// TwinCAT 3 PLC project PRG_B_HMIManager
// Title: B_HMIManager
// Company: RafałOS
// Author: Rafał Osajda
// ProjectVersion: 0.0.0.21
// ProgramVersion: 3.1.4024.0
// libraries:
//   B_Base, * (RafalOS)
//   B_Base_HMI_Connector, * (RafalOS)
//   B_HMIElements, * (RafalOS)
//   B_MachineControl, * (RafalOS)
//   B_MachineControl_HMI_Connector, * (RafalOS)
//   B_StatesAndModes, * (RafalOS)
//   Tc2_Standard, * (Beckhoff Automation GmbH)
//   Tc2_System, * (Beckhoff Automation GmbH)
//   Tc3_Module, * (Beckhoff Automation GmbH)
// project tree:
//   / PlcTask.TcTTO
//   POUs Compilation/ PRG_Compilation.TcPOU (not stored)
//   POUs/01_HMIManager/ FB_HMIManager.TcPOU, ITF_HMIManager.TcIO (not stored), ITF_HMIManagerConfigure.TcIO, ST_HMIManager.TcDUT
//   POUs/02_Configuration/ FB_HMIConfigure.TcPOU, ITF_HMIConfiguration.TcIO, ITF_HMIConfigure.TcIO (not stored)
// real-time tasks:
//   TASK PlcTask: cycle T#10ms, priority 20, ADS port 350

CONFIGURATION PRG_B_HMIManager
    RESOURCE PLC ON TwinCAT3
        TASK PlcTask(INTERVAL := T#10ms, PRIORITY := 20);
        PROGRAM PRG_Compilation WITH PlcTask : PRG_Compilation;
    END_RESOURCE
END_CONFIGURATION

// ---- POUs/01_HMIManager/ST_HMIManager.TcDUT
TYPE ST_HMIManager EXTENDS ST_BaseGroupElement_HMI_Link :
STRUCT
	stMainMenu			: ST_HMIEMenu_HMI_Link;
	stMachineControl	: ST_MCHMIMachineControl_HMI_Link;
	stRecipe			: ST_BaseRecipe_HMI;
END_STRUCT
END_TYPE

// ---- POUs/01_HMIManager/ITF_HMIManagerConfigure.TcIO
INTERFACE ITF_HMIManagerConfigure EXTENDS ITF_Base

(*			
	RafalOS
	Rafał Osajda		07.12.2025		TC 4024.66
	Dodawanie elementów do systemmu wyświetlania
*)
METHOD AddElementFromConfiguration
VAR_INPUT
	fbTopElementHMI		: ITF_BaseTopElement_HMI;
END_VAR
END_METHOD

(*			
	RafalOS
	Rafał Osajda		20.11.2025		TC 4024.66
	Dodawanie rozszerzonego wyświetlania danych inna prezenacja danych niż domyślna lista
*)
METHOD PUBLIC AddExtendedDisplayToPrepScrModuleFromConfiguration : BOOL
VAR_INPUT
	itfModule		: ITF_MCHMIPrepareDataForScreenExtension;
	itfExtension	: ITF_MCHMIDisplayExtension;
END_VAR
END_METHOD

(*			
	RafalOS
	Rafał Osajda		19.11.2025		TC 4024.66
	Dodanie połączenia do MachineControl  wywoływane z konfiguracji
*)
METHOD AddMachineControlConnectorFromConfiguration : BOOL
VAR_INPUT
	itfMachineControl	: ITF_MCHMIMachineControl_HMI;
END_VAR
END_METHOD

(*			
	RafalOS
	Rafał Osajda		14.11.2025		TC 4024.66
	Dodanie do systemu menu głównego 
*)
METHOD PUBLIC AddMainMenuFromConfiguration : BOOL
VAR_INPUT
	fbMenu			: ITF_HMIEMenu;
	fbMenu_HMI		: ITF_HMIEMenu_HMI;
END_VAR
END_METHOD

(*			
	RafalOS
	Rafał Osajda		19.11.2025		TC 4024.66
	Dodanie modułów do przygotowywania stron do wyświetlenia
*)
METHOD AddPrepareScreenModuleFromConfiguration : BOOL
VAR_INPUT
	itfModule	: ITF_MCHMIPrepareScreen_Init;
END_VAR
END_METHOD

(*			
	RafalOS
	Rafał Osajda		26.11.2025		TC 4024.66
	Podłaczenie modułu receptur
*)
METHOD PUBLIC AddRecipeModuleFromConfiguration : BOOL
VAR_INPUT
	fbRecipeModule		: ITF_BaseRecipe_HMI;
END_VAR
END_METHOD

METHOD PUBLIC GetNumberOfAddedButtons : INT
VAR_INPUT
END_VAR
END_METHOD

(*			
	RafalOS
	Rafał Osajda		18.11.2025		TC 4024.66
	Podłączenie głównej struktury danych dla domyślnych elementów 
*)
METHOD LinkHMIManagerDataFromConfiguration : BOOL
VAR_INPUT
	stData					: REFERENCE TO ST_HMIManager;
END_VAR
END_METHOD

METHOD PUBLIC LinkPrepareScreenToArrayFromConfiguration : BOOL
VAR_INPUT
	iScreen		: INT;
	iMode		: INT;
	itfModule	: ITF_MCHMIPrepareDataForScreen;
END_VAR
END_METHOD

(*			
	RafalOS
	Rafał Osajda		13.11.2025		TC 4024.66
	Podłączenie wsyzstkich zmiennych pochodzących od Programu safety 
*)
METHOD PUBLIC LinkSafetyToaddedElementsFromConfiguration : BOOL
VAR_INPUT
	flSS1				: ITF_BaseFlagGet;
	flSTO				: ITF_BaseFlagGet;
END_VAR
END_METHOD

(*			
	RafalOS
	Rafał Osajda		18.11.2025		TC 4024.66
	Ustawia przycisk na aktywny  - pierwsze okno w wyświetlaniu wizualizacji - wywoływane z konfiguracji
*)
METHOD SetButtonActiveFromConfiguration : BOOL
VAR_INPUT
	iNumber		: INT;	//numr przycisku
	bValue		: BOOL;
END_VAR
END_METHOD

(*			
	RafalOS
	Rafał Osajda		18.11.2025		TC 4024.66
	Ustawia przyciski na wlaczone lub wylaczone - możliwośc naciśnięcia
*)
METHOD SetButtonsEnabledFromConfiguration : BOOL
VAR_INPUT
	iNumber		: INT;	//numr przycisku
	bValue		: BOOL;
END_VAR
END_METHOD

(*			
	RafalOS
	Rafał Osajda		18.11.2025		TC 4024.66
	Ustawia przyciski na widoczne lub nie widoczne
*)
METHOD SetButtonsVisibleFromConfiguration : BOOL
VAR_INPUT
	iNumber		: INT;	//numr przycisku
	bValue		: BOOL;
END_VAR
END_METHOD

END_INTERFACE

// ---- POUs/02_Configuration/ITF_HMIConfiguration.TcIO
INTERFACE ITF_HMIConfiguration

(*			
	RafalOS
	Rafał Osajda		07.12.2025		TC 4024.66
	Dodawanie elementów do systemmu wyświetlania
*)
METHOD AddElement
VAR_INPUT
	itfHMIManager	: ITF_HMIManagerConfigure;
END_VAR
END_METHOD

(*			
	RafalOS
	Rafał Osajda		20.11.2025		TC 4024.66
	Dodawanie rozszerzonego wyświetlania danych inna prezenacja danych niż domyślna lista
*)
METHOD PUBLIC AddExtendedDisplayToPrepScrModule : BOOL
VAR_INPUT
	itfHMIManager	: ITF_HMIManagerConfigure;
END_VAR
END_METHOD

(*			
	RafalOS
	Rafał Osajda		19.11.2025		TC 4024.66
	Dodanie połączenia do MachineControl
*)
METHOD AddMachineControlConnector : BOOL
VAR_INPUT
	itfHMIManager	: ITF_HMIManagerConfigure;
END_VAR
END_METHOD

(*			
	RafalOS
	Rafał Osajda		14.11.2025		TC 4024.66
	Dodanie do systemu menu głównego 
*)
METHOD PUBLIC AddMainMenu : BOOL
VAR_INPUT
	itfHMIManager	: ITF_HMIManagerConfigure;
END_VAR
END_METHOD

(*			
	RafalOS
	Rafał Osajda		19.11.2025		TC 4024.66
	Dodanie modułów do przygotowywania stron do wyświetlenia
*)
METHOD AddPrepareScreenModule : BOOL
VAR_INPUT
	itfHMIManager	: ITF_HMIManagerConfigure;
END_VAR
END_METHOD

(*			
	RafalOS
	Rafał Osajda		26.11.2025		TC 4024.66
	Podłaczenie modułu receptur
*)
METHOD PUBLIC AddRecipeModule : BOOL
VAR_INPUT
	itfHMIManager	: ITF_HMIManagerConfigure;
END_VAR
END_METHOD

(*			
	RafalOS
	Rafał Osajda		18.11.2025		TC 4024.66
	Podłączenie głównej struktury danych dla domyślnych elementów 
*)
METHOD LinkHMIManagerData : BOOL
VAR_INPUT
	itfHMIManager	: ITF_HMIManagerConfigure;
END_VAR
END_METHOD

(*			
	RafalOS
	Rafał Osajda		16.12.2025		TC 4024.66
	Wywołanie linkowania zmiennych w topelemencie i jego dzieciach
*)
METHOD PUBLIC LinkMachineData : BOOL
VAR_INPUT
	itfHMIManager	: ITF_HMIManagerConfigure;
END_VAR
END_METHOD

(*			
	RafalOS
	Rafał Osajda		13.11.2025		TC 4024.66
	Podłączenie wsyzstkich zmiennych pochodzących od Programu safety 
*)
METHOD PUBLIC LinkSafetyToaddedElements : BOOL
VAR_INPUT
	itfHMIManager	: ITF_HMIManagerConfigure;
END_VAR
END_METHOD

(*			
	RafalOS
	Rafał Osajda		18.11.2025		TC 4024.66
	Ustawia przycisk na aktywny  - pierwsze okno w wyświetlaniu wizualizacji
*)
METHOD SetButtonActive : BOOL
VAR_INPUT
	itfHMIManager	: ITF_HMIManagerConfigure;
END_VAR
END_METHOD

(*			
	RafalOS
	Rafał Osajda		18.11.2025		TC 4024.66
	Ustawia przyciski na wlaczone lub wylaczone - możliwośc naciśnięcia
*)
METHOD SetButtonsEnabled : BOOL
VAR_INPUT
	itfHMIManager	: ITF_HMIManagerConfigure;
END_VAR
END_METHOD

(*			
	RafalOS
	Rafał Osajda		18.11.2025		TC 4024.66
	Ustawia przyciski na widoczne lub nie widoczne
*)
METHOD SetButtonsVisible : BOOL
VAR_INPUT
	itfHMIManager	: ITF_HMIManagerConfigure;
END_VAR
END_METHOD

END_INTERFACE

// ---- POUs/01_HMIManager/FB_HMIManager.TcPOU
FUNCTION_BLOCK FB_HMIManager EXTENDS FB_BaseGroupElement IMPLEMENTS ITF_HMIManager, ITF_HMIManagerConfigure
VAR
	(*	Inicjalizacja		*)
	bInitializeCycle			: BOOL;
	bInitDone					: BOOL;
	bIsValidData				: bool;
	(*	Konfiguracja		*)
	itfHMIConfigure				: ITF_HMIConfigure;		//moduł konfiguracji
	(*	Menu główne	*)
	itfMainMenu					: ITF_HMIEMenu;
	itfMainMenuHMI				: ITF_HMIEMenu_HMI;
	iNumberOfButtonMainMenu		: INT;
	iNumberOfActiveScreen		: INT;
	iNumberOfPreviewScreen		: INT;
	bChangePage					: BOOL;
//	(*	Obsługa zmiany strony	*)
//	arrChangePageSupport		: ARRAY [0..GVL_HMIEConstans.MAX_NUMBER_OF_BUTTON_IN_MENU] OF 
//									ARRAY [0..GVL_SaMConstans.NUMBER_OF_MODES] OF ITF_PrepareDataForScreen;
	(*	Dana wspólne dla całego systemu	*)
	refstManagerData			: REFERENCE TO ST_HMIManager;
	(*	Łącznik do MachineControl	*)
	itfMachineControl			: ITF_MCHMIMachineControl_HMI;
	(*	Lista dodanych elementów	*)
	stElement					: ST_ListOfElement_HMI;
END_VAR

IF (NOT THIS^.bInitializeCycle) THEN
	THIS^.bInitializeCycle		:= TRUE;
	THIS^.bInitDone				:= THIS^.InitializeCycle ();
ELSIF (THIS^.bInitDone) THEN
	THIS^.ExecuteCycle ();
END_IF

(*			
	RafalOS
	Rafał Osajda		07.12.2025		TC 4024.66
	Dodawanie elementów do systemmu wyświetlania
*)
METHOD AddElementFromConfiguration
VAR_INPUT
	fbTopElementHMI		: ITF_BaseTopElement_HMI;
END_VAR
fbTopElementHMI.JoinTheList (
	refstList		:= THIS^.stElement,
	iNumberOfParent := 0
);

fbTopElementHMI.LinkCommonData (stCommonData := THIS^.refstCommonData);
END_METHOD

(*			
	RafalOS
	Rafał Osajda		20.11.2025		TC 4024.66
	Dodawanie rozszerzonego wyświetlania danych inna prezenacja danych niż domyślna lista
*)
METHOD PUBLIC AddExtendedDisplayToPrepScrModuleFromConfiguration : BOOL
VAR_INPUT
	itfModule		: ITF_MCHMIPrepareDataForScreenExtension;
	itfExtension	: ITF_MCHMIDisplayExtension;
END_VAR
itfModule.LinkExtensionDisplay (fbExtendedDisplay := itfExtension);
END_METHOD

(*			
	RafalOS
	Rafał Osajda		19.11.2025		TC 4024.66
	Dodanie połączenia do MachineControl  wywoływane z konfiguracji
*)
METHOD AddMachineControlConnectorFromConfiguration : BOOL
VAR_INPUT
	itfMachineControl	: ITF_MCHMIMachineControl_HMI;
END_VAR
THIS^.itfMachineControl := itfMachineControl;

THIS^.itfMachineControl.LinkCommonData (stCommonData := THIS^.refstCommonData);
END_METHOD

(*			
	RafalOS
	Rafał Osajda		14.11.2025		TC 4024.66
	Dodanie do systemu menu głównego 
*)
METHOD PUBLIC AddMainMenuFromConfiguration : BOOL
VAR_INPUT
	fbMenu			: ITF_HMIEMenu;
	fbMenu_HMI		: ITF_HMIEMenu_HMI;
END_VAR
THIS^.SetText (eLocation := E_BaseLocation.pl, wsDescription := "Menu główne");
THIS^.SetText (eLocation := E_BaseLocation.en, wsDescription := "Main menu");
THIS^.SetText (eLocation := E_BaseLocation.de, wsDescription := "Hauptmenü");
fbMenu.SetName (stName := THIS^.GetTexts ());
THIS^.AddControlElement (itfControlElement := fbMenu);

THIS^.itfMainMenu := fbMenu;
THIS^.itfMainMenu.LinkCommonData (stCommonData := THIS^.refstCommonData);
//THIS^.itfMainMenu.LinkSS1 (fbSS1 := THIS^.itfSS1);
//THIS^.itfMainMenu.LinkSTO (fbSTO := THIS^.itfSTO);

THIS^.itfMainMenuHMI  := fbMenu_HMI;
THIS^.itfMainMenuHMI.LinkCommonData (stCommonData := THIS^.refstCommonData);
END_METHOD

(*			
	RafalOS
	Rafał Osajda		29.10.2025		TC 4024.66
	Dodawanie intefejsu konfiguracji
*)
METHOD PUBLIC AddModulConfigure : BOOL
VAR_INPUT
	fbHMIConfigure			: ITF_HMIConfigure;
END_VAR
THIS^.itfHMIConfigure		:= fbHMIConfigure;
END_METHOD

(*			
	RafalOS
	Rafał Osajda		19.11.2025		TC 4024.66
	Dodanie modułów do przygotowywania stron do wyświetlenia
*)
METHOD AddPrepareScreenModuleFromConfiguration : BOOL
VAR_INPUT
	itfModule	: ITF_MCHMIPrepareScreen_Init;
END_VAR
THIS^.itfMachineControl.AddPrepareScreenModuleFromManager (
	itfModule	:= itfModule
);
itfModule.LinkCommonData (stCommonData := THIS^.refstCommonData);
END_METHOD

(*			
	RafalOS
	Rafał Osajda		26.11.2025		TC 4024.66
	Podłaczenie modułu receptur
*)
METHOD PUBLIC AddRecipeModuleFromConfiguration : BOOL
VAR_INPUT
	fbRecipeModule		: ITF_BaseRecipe_HMI;
END_VAR
THIS^.itfMachineControl.AddRecipeModulFormManager (fbRecipeModul := fbRecipeModule);
END_METHOD

(*			
	RafalOS
	Rafał Osajda		10.11.2025		TC 4024.66
	Główna metoda sterujaca wyświetlaniem dsanych na HMI
*)
METHOD PUBLIC ExecuteCycle
	(* Testowanie MenuGlownego	*)
THIS^.itfMainMenu.Testing ();
	(*	Przepisanie Aktualnych zmiennych menu do struktury danych HMI	*)

THIS^.itfMainMenuHMI.PrepareDataForHMI ();
	
	(*	Aktualizacja zmiennych przy zmianie strony	*)
THIS^.bChangePage := THIS^.itfMainMenuHMI.IsChangePage ();
THIS^.refstManagerData.stMachineControl.stCommonData.bChangePage := THIS^.bChangePage;

	(*	Test wybranej receptury	*)
THIS^.itfMachineControl.GetInformationLatestRecipes ();

IF (THIS^.bChangePage) THEN
	(*	Skasowanie flagi zmiany strony	*)
	THIS^.itfMainMenu.ResetChangePage ();
	THIS^.iNumberOfPreviewScreen := THIS^.itfMainMenuHMI.GetNumberOfPreviewScreen ();
	THIS^.iNumberOfActiveScreen := THIS^.itfMainMenuHMI.GetNumberOfActiveScreen ();
	
	
	THIS^.itfMachineControl.ClearAfterScreenFroHMIManager (
		iScreen	:= THIS^.iNumberOfPreviewScreen,
		iMode	:= THIS^.itfMachineControl.GetActiveModeFromManager ()
	);
	THIS^.itfMachineControl.PrepareForScreenFromHMIManager (
		iScreen	:= THIS^.iNumberOfActiveScreen,
		iMode	:= THIS^.itfMachineControl.GetActiveModeFromManager ()
	);
END_IF

	(*	Odświerzenia strrony 	*)
THIS^.itfMachineControl.PrepareDataForScreenFromHMIManager (
	iScreen	:= THIS^.iNumberOfActiveScreen,
	iMode	:= THIS^.itfMachineControl.GetActiveModeFromManager ()
);
END_METHOD

METHOD FB_init : BOOL
VAR_INPUT
	bInitRetains : BOOL; // if TRUE, the retain variables are initialized (warm start / cold start)
	bInCopyCode : BOOL;  // if TRUE, the instance afterwards gets moved into the copy code (online change)
END_VAR
THIS^.SetText (eLocation := E_BaseLocation.pl, wsDescription := "HMI Menadżer");
THIS^.SetText (eLocation := E_BaseLocation.en, wsDescription := "HMI Manager");
THIS^.SetText (eLocation := E_BaseLocation.de, wsDescription := "HMI Manager");
THIS^.SetName (stName := THIS^.GetTexts ());
END_METHOD

METHOD PUBLIC GetNumberOfAddedButtons : INT
VAR_INPUT
END_VAR
GetNumberOfAddedButtons := THIS^.itfMainMenu.GetNumberOfAddedButton ();
END_METHOD

METHOD PRIVATE InitializeCycle : BOOL
VAR
	bResult					: BOOL;
	iI: INT;
END_VAR
bResult				:= TRUE;

bResult				:= bResult AND THIS^.itfHMIConfigure.Configure (fbHMIManager := THIS^);

InitializeCycle		:= bResult;
END_METHOD

(*			
	RafalOS
	Rafał Osajda		18.11.2025		TC 4024.66
	Podłączenie głównej struktury danych dla domyślnych elementów 
*)
METHOD LinkHMIManagerDataFromConfiguration : BOOL
VAR_INPUT
	stData					: REFERENCE TO ST_HMIManager;
END_VAR
THIS^.refstManagerData	REF= stData;

THIS^.itfMainMenuHMI.LinkHMIEMenuData (stData := stData.stMainMenu);

THIS^.itfMachineControl.LinkMachineControlData (stData := stData.stMachineControl);

IF (__ISVALIDREF (THIS^.refstManagerData)) THEN
	THIS^.bIsValidData := TRUE;
	LinkHMIManagerDataFromConfiguration := TRUE;
END_IF
END_METHOD

METHOD PUBLIC LinkPrepareScreenToArrayFromConfiguration : BOOL
VAR_INPUT
	iScreen		: INT;
	iMode		: INT;
	itfModule	: ITF_MCHMIPrepareDataForScreen;
END_VAR
THIS^.itfMachineControl.LinkPrepareScreenToArrayFromConfiguration (
	iScreen		:= iScreen,
	iMode		:= iMode,
	itfModule	:= itfModule
);
END_METHOD

(*			
	RafalOS
	Rafał Osajda		13.11.2025		TC 4024.66
	Podłączenie wsyzstkich zmiennych pochodzących od Programu safety 
*)
METHOD PUBLIC LinkSafetyToaddedElementsFromConfiguration : BOOL
VAR_INPUT
	flSS1				: ITF_BaseFlagGet;
	flSTO				: ITF_BaseFlagGet;
END_VAR
THIS^.LinkSS1 (fbSS1 := flSS1);
THIS^.LinkSTO (fbSTO := flSTO);
END_METHOD

(*			
	RafalOS
	Rafał Osajda		18.11.2025		TC 4024.66
	Ustawia przycisk na aktywny  - pierwsze okno w wyświetlaniu wizualizacji - wywoływane z konfiguracji
*)
METHOD SetButtonActiveFromConfiguration : BOOL
VAR_INPUT
	iNumber		: INT;	//numr przycisku
	bValue		: BOOL;
END_VAR
THIS^.itfMainMenu.SetActiveButton (iButton := iNumber, bIN := bValue);
END_METHOD

(*			
	RafalOS
	Rafał Osajda		18.11.2025		TC 4024.66
	Ustawia przyciski na wlaczone lub wylaczone - możliwośc naciśnięcia
*)
METHOD SetButtonsEnabledFromConfiguration : BOOL
VAR_INPUT
	iNumber		: INT;	//numr przycisku
	bValue		: BOOL;
END_VAR
THIS^.itfMainMenu.SetEnableButton (iButton := iNumber, bIN := bValue);
END_METHOD

(*			
	RafalOS
	Rafał Osajda		18.11.2025		TC 4024.66
	Ustawia przyciski na widoczne lub nie widoczne
*)
METHOD SetButtonsVisibleFromConfiguration : BOOL
VAR_INPUT
	iNumber		: INT;	//numr przycisku
	bValue		: BOOL;
END_VAR
THIS^.itfMainMenu.SetVisibleButton (iButton := iNumber, bIN := bValue);
END_METHOD

END_FUNCTION_BLOCK

// ---- POUs/02_Configuration/FB_HMIConfigure.TcPOU
FUNCTION_BLOCK FB_HMIConfigure EXTENDS FB_Base IMPLEMENTS ITF_HMIConfigure
VAR
	(*	Baza konfiguracji	*)
	arritfConfigure				: ARRAY [1..10] OF ITF_HMIConfiguration;
	iNubmerOfAddedConfigure		: INT;
END_VAR

METHOD PUBLIC AddConfiguration : BOOL
VAR_INPUT
	fbConfigure		: ITF_HMIConfiguration;
END_VAR
IF (THIS^.iNubmerOfAddedConfigure + 1 <= 10) THEN
	THIS^.iNubmerOfAddedConfigure	:= THIS^.iNubmerOfAddedConfigure + 1;
	THIS^.arritfConfigure [THIS^.iNubmerOfAddedConfigure]	:= fbConfigure;
	AddConfiguration	:= TRUE;
ELSE
	AddConfiguration	:= FALSE;
END_IF
END_METHOD

METHOD PUBLIC Configure : BOOL
VAR_INPUT
	fbHMIManager			: ITF_HMIManagerConfigure;
END_VAR
VAR
	bResult				: BOOL;
	iI					: INT;
END_VAR
bResult			:= TRUE;

THIS^.arritfConfigure [1].AddMainMenu (itfHMIManager := fbHMIManager);
THIS^.arritfConfigure [1].AddMachineControlConnector (itfHMIManager := fbHMIManager);
THIS^.arritfConfigure [1].AddPrepareScreenModule (itfHMIManager := fbHMIManager);
THIS^.arritfConfigure [1].AddExtendedDisplayToPrepScrModule (itfHMIManager := fbHMIManager);
this^.arritfConfigure [1].AddRecipeModule (itfHMIManager := fbHMIManager);
	
FOR iI := 1 TO THIS^.iNubmerOfAddedConfigure DO 
	IF (THIS^.arritfConfigure [iI] <> 0) THEN
		THIS^.arritfConfigure [iI].SetButtonActive (itfHMIManager	:= fbHMIManager);
		THIS^.arritfConfigure [iI].SetButtonsVisible (itfHMIManager	:= fbHMIManager);
		THIS^.arritfConfigure [iI].SetButtonsEnabled (itfHMIManager	:= fbHMIManager);
		THIS^.arritfConfigure [iI].AddElement (itfHMIManager	:= fbHMIManager);
		THIS^.arritfConfigure [iI].LinkMachineData (itfHMIManager	:= fbHMIManager);
		
	END_IF
END_FOR
THIS^.arritfConfigure [1].LinkSafetyToaddedElements (itfHMIManager := fbHMIManager);
THIS^.arritfConfigure [1].LinkHMIManagerData (itfHMIManager := fbHMIManager);

Configure		:= bResult;
END_METHOD

END_FUNCTION_BLOCK
